VAR_GLOBAL
	MEASUREMENT_ANGLE : UINT := 1;
	HEIGHT_VIRTUAL : UINT:= 2;
	HEIGHT : UINT := 3;
	HORIZONTAL : UINT := 4;
	HORIZONTAL_VIRTUAL : UINT := 5;
	ROTATION_VIRTUAL : UINT := 6;
	ROTATION_LINEAR_REAL : UINT := 7;
	ROTATION_LINEAR_VIRTUAL_ENCODER : UINT := 8; //Encoder only axis to get speed information from
END_VAR

(* stored: Version 1.1.0.1, ProductVersion 3.1.4026.12
   GVL GVL_AxisNames: Id {ac2d037b-2b8c-41f4-8d85-bcb635f10da5} *)
